(* Schneider Machine Expert - Basic project TMA0070_BOTTOM CASE SCREWING, file version 2.8.0.0 *)
(* ProjectInformations: Name=New project *)

HARDWARE
  Cpu 0: TM221CE16T
  EthernetConfiguration: NetworkName=M221, IpAllocationMode=FixedAddress, IpAddress=192.168.0.150, SubnetMask=255.255.255.0
  SerialLineConfiguration: Baud=Baud19200, Parity=ParityEven, DataBits=DataBits8, StopBits=StopBits1, PhysicalMedium=PhysicalMediumRs485, TransmissionMode=TransmissionModeModbusRtu, SlaveId=1, Addressing=SlaveAddressing
  MastTask: UsePeriodScanMode=false, PeriodScan=100
  FastTask: Period=255
  CpuBehavior: StartingMode=StartAsPreviousState, AutoSaveRamOnEeprom=true, WatchdogPeriod=250

SYMBOLS  (address, symbol, comment, settings)
  %M20      IB_ESTOP
  %M21      IB_CYL  "TURUNSTART"
  %M23      IB_TIMER
  %M27      VALID_BARCODE
  %M28      INVALID_BARCODE
  %M29      IB_TRIGGER_KEYENCE
  %M32      MACHINE_RUNNING
  %M33      ERROR_BARCODE
  %M34      SAFETY_TRIGGER
  %M35      TURUNDONE_SENSOR_TURUN
  %M80      PASS
  %TM0        [Preset=2, Base=OneSecond]
  %TM1        [Preset=2, Base=OneSecond]
  %I0.0     ESTOP
  %I0.1     START_PB
  %I0.2     RESET_PB
  %I0.3     CURTAIN  "CURTAIN SENSOR"
  %I0.4     C_NEWTON  "CHECK OUTX LOAD CELL"
  %I0.5     TIMER  "TIMER DONE"
  %I0.6     RS_CYL_UP
  %I0.7     RS_CYL_DOWN
  %Q0.0     CYL_PRESS
  %Q0.1     START_TIIMER
  %Q0.2     TRIGGER_KEYENCE
  %Q0.3     RED_LIGHT
  %Q0.4     YELLOW_LIGHT_
  %Q0.5     GREEN_LIGHT
  %IW0.0      [Type=Type_0_10V, Scope=Scope_Normal, Minimum=0, Maximum=1000]

POU SEQUENCE
  (* SectionNumber=1 *)

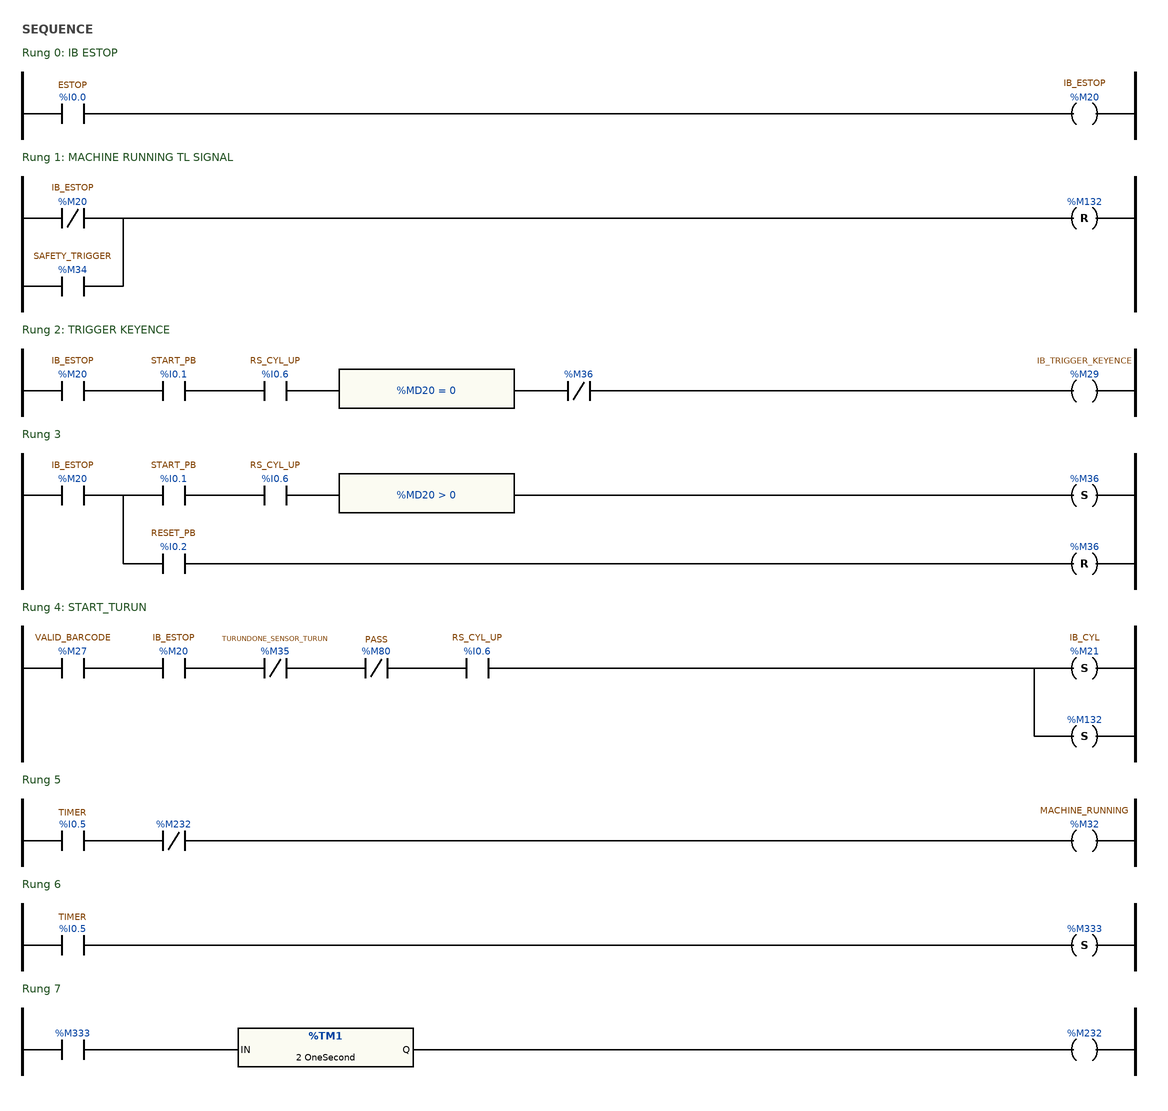

// Rung 0: IB ESTOP
  LD %I0.0                (* ESTOP *)
  ST %M20                 (* IB_ESTOP *)
  // as ST:
  //   IB_ESTOP := ESTOP;

// Rung 1: MACHINE RUNNING TL SIGNAL
  LDN %M20                (* IB_ESTOP *)
  OR %M34                 (* SAFETY_TRIGGER *)
  R %M132
  // as ST:
  //   IF NOT IB_ESTOP OR SAFETY_TRIGGER THEN %M132 := FALSE; END_IF;

// Rung 2: TRIGGER KEYENCE
  LD %M20                 (* IB_ESTOP *)
  AND %I0.1               (* START_PB *)
  AND %I0.6               (* RS_CYL_UP *)
  AND [ %MD20 = 0 ]
  ANDN %M36
  ST %M29                 (* IB_TRIGGER_KEYENCE *)
  // as ST:
  //   IB_TRIGGER_KEYENCE := IB_ESTOP AND START_PB AND RS_CYL_UP AND %MD20 = 0 AND NOT %M36;

// Rung 3
  LD %M20                 (* IB_ESTOP *)
  MPS
  AND %I0.1               (* START_PB *)
  AND %I0.6               (* RS_CYL_UP *)
  AND [ %MD20 > 0 ]
  S %M36
  MPP
  AND %I0.2               (* RESET_PB *)
  R %M36
  // as ST:
  //   IF IB_ESTOP AND START_PB AND RS_CYL_UP AND %MD20 > 0 THEN %M36 := TRUE; END_IF;
  //   IF IB_ESTOP AND RESET_PB THEN %M36 := FALSE; END_IF;

// Rung 4: START_TURUN
  LD %M27                 (* VALID_BARCODE *)
  AND %M20                (* IB_ESTOP *)
  ANDN %M35               (* TURUNDONE_SENSOR_TURUN *)
  ANDN %M80               (* PASS *)
  AND %I0.6               (* RS_CYL_UP *)
  S %M21                  (* IB_CYL *)
  S %M132
  // as ST:
  //   IF VALID_BARCODE AND IB_ESTOP AND NOT TURUNDONE_SENSOR_TURUN AND NOT PASS AND RS_CYL_UP THEN IB_CYL := TRUE; END_IF;
  //   IF VALID_BARCODE AND IB_ESTOP AND NOT TURUNDONE_SENSOR_TURUN AND NOT PASS AND RS_CYL_UP THEN %M132 := TRUE; END_IF;

// Rung 5
  LD %I0.5                (* TIMER *)
  ANDN %M232
  ST %M32                 (* MACHINE_RUNNING *)
  // as ST:
  //   MACHINE_RUNNING := TIMER AND NOT %M232;

// Rung 6
  LD %I0.5                (* TIMER *)
  S %M333
  // as ST:
  //   IF TIMER THEN %M333 := TRUE; END_IF;

// Rung 7
  BLK %TM1
  LD %M333
  IN
  OUT_BLK
  LD Q
  ST %M232
  END_BLK
  // as ST:
  //   %TM1(IN := %M333);
  //   %M232 := %TM1.Q;

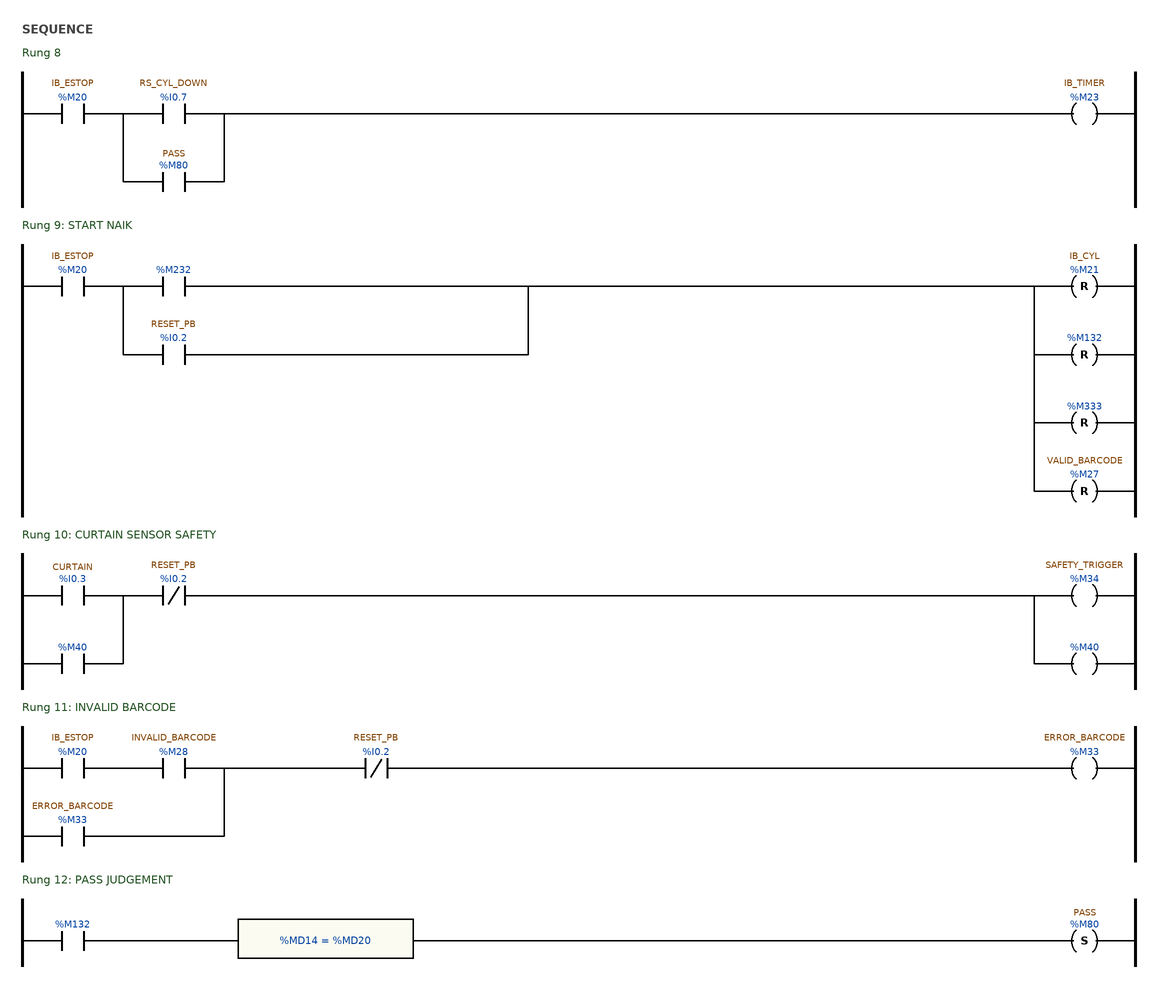

// Rung 8
  LD %M20                 (* IB_ESTOP *)
  AND( %I0.7              (* RS_CYL_DOWN *)
  OR %M80                 (* PASS *)
  )
  ST %M23                 (* IB_TIMER *)
  // as ST:
  //   IB_TIMER := IB_ESTOP AND (RS_CYL_DOWN OR PASS);

// Rung 9: START NAIK
  LD %M20                 (* IB_ESTOP *)
  AND( %M232
  OR %I0.2                (* RESET_PB *)
  )
  R %M21                  (* IB_CYL *)
  R %M132
  R %M333
  R %M27                  (* VALID_BARCODE *)
  // as ST:
  //   IF IB_ESTOP AND (%M232 OR RESET_PB) THEN IB_CYL := FALSE; END_IF;
  //   IF IB_ESTOP AND (%M232 OR RESET_PB) THEN %M132 := FALSE; END_IF;
  //   IF IB_ESTOP AND (%M232 OR RESET_PB) THEN %M333 := FALSE; END_IF;
  //   IF IB_ESTOP AND (%M232 OR RESET_PB) THEN VALID_BARCODE := FALSE; END_IF;

// Rung 10: CURTAIN SENSOR SAFETY
  LD %I0.3                (* CURTAIN *)
  OR %M40
  ANDN %I0.2              (* RESET_PB *)
  ST %M34                 (* SAFETY_TRIGGER *)
  ST %M40
  // as ST:
  //   SAFETY_TRIGGER := (CURTAIN OR %M40) AND NOT RESET_PB;
  //   %M40 := (CURTAIN OR %M40) AND NOT RESET_PB;

// Rung 11: INVALID BARCODE
  LD %M20                 (* IB_ESTOP *)
  AND %M28                (* INVALID_BARCODE *)
  OR %M33                 (* ERROR_BARCODE *)
  ANDN %I0.2              (* RESET_PB *)
  ST %M33                 (* ERROR_BARCODE *)
  // as ST:
  //   ERROR_BARCODE := (IB_ESTOP AND INVALID_BARCODE OR ERROR_BARCODE) AND NOT RESET_PB;

// Rung 12: PASS JUDGEMENT
  LD %M132
  AND [ %MD14 = %MD20 ]
  S %M80                  (* PASS *)
  // as ST:
  //   IF %M132 AND %MD14 = %MD20 THEN PASS := TRUE; END_IF;

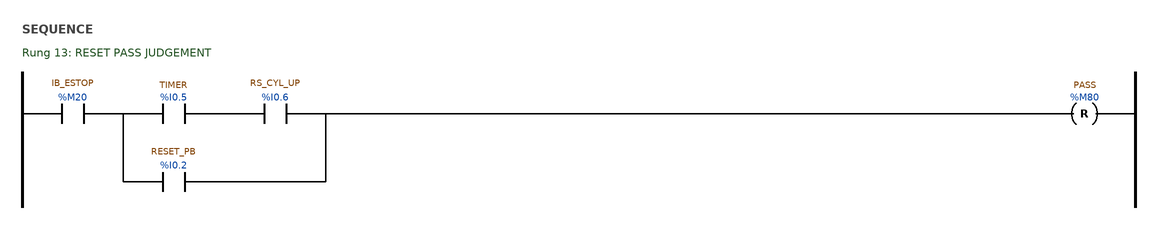

// Rung 13: RESET PASS JUDGEMENT
  LD %M20                 (* IB_ESTOP *)
  AND( %I0.5              (* TIMER *)
  AND %I0.6               (* RS_CYL_UP *)
  OR %I0.2                (* RESET_PB *)
  )
  R %M80                  (* PASS *)
  // as ST:
  //   IF IB_ESTOP AND (TIMER AND RS_CYL_UP OR RESET_PB) THEN PASS := FALSE; END_IF;

POU I/0
  (* SectionNumber=2 *)

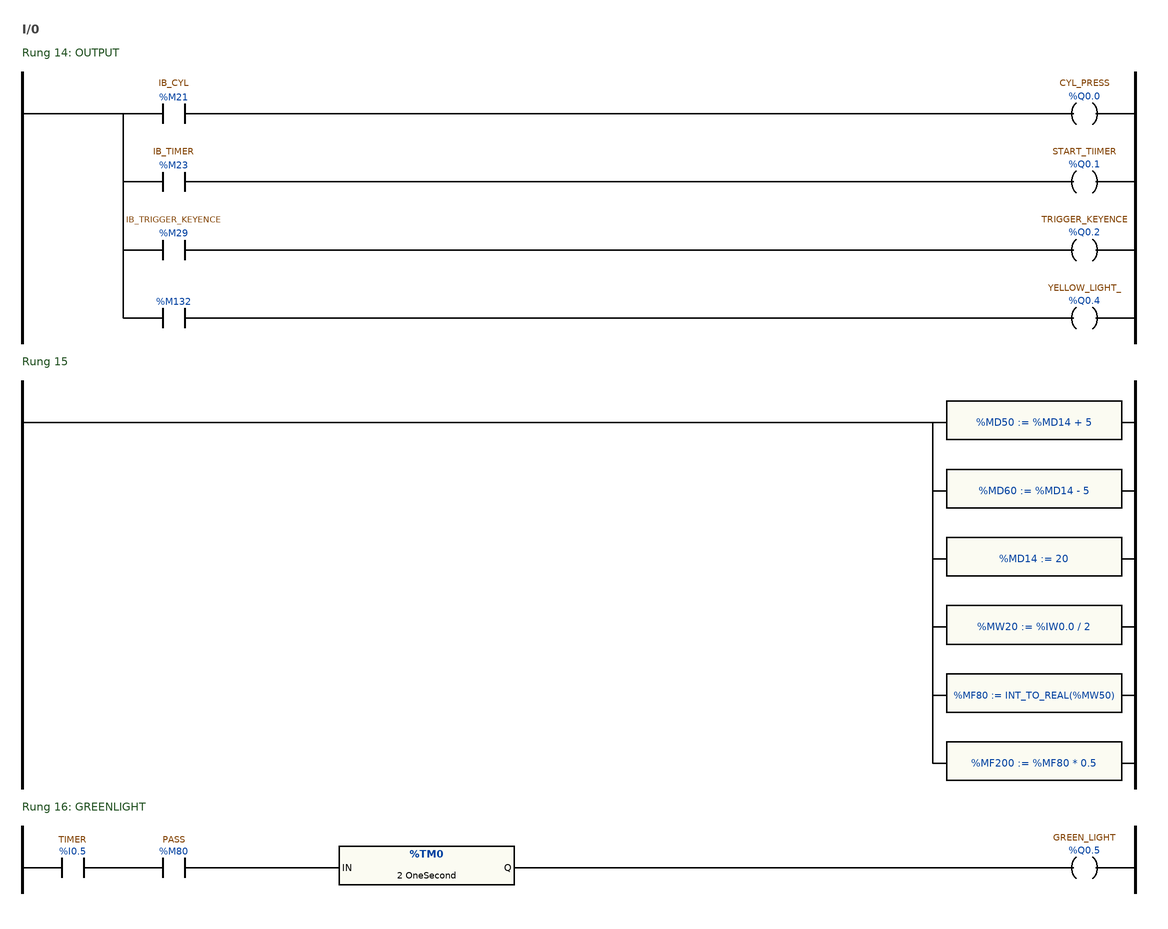

// Rung 14: OUTPUT
  LD 1
  MPS
  AND %M21                (* IB_CYL *)
  ST %Q0.0                (* CYL_PRESS *)
  MRD
  AND %M23                (* IB_TIMER *)
  ST %Q0.1                (* START_TIIMER *)
  MRD
  AND %M29                (* IB_TRIGGER_KEYENCE *)
  ST %Q0.2                (* TRIGGER_KEYENCE *)
  MPP
  AND %M132
  ST %Q0.4                (* YELLOW_LIGHT_ *)
  // as ST:
  //   CYL_PRESS := IB_CYL;
  //   START_TIIMER := IB_TIMER;
  //   TRIGGER_KEYENCE := IB_TRIGGER_KEYENCE;
  //   YELLOW_LIGHT_ := %M132;

// Rung 15
  LD 1
  [ %MD50 := %MD14 + 5 ]
  [ %MD60 := %MD14 - 5 ]
  [ %MD14 := 20 ]
  [ %MW20 := %IW0.0 / 2 ]
  [ %MF80 := INT_TO_REAL ( %MW50 ) ]
  [ %MF200 := %MF80 * 0.5 ]
  // as ST:
  //   %MD50 := %MD14 + 5;
  //   %MD60 := %MD14 - 5;
  //   %MD14 := 20;
  //   %MW20 := %IW0.0 / 2;
  //   %MF80 := INT_TO_REAL ( %MW50 );
  //   %MF200 := %MF80 * 0.5;

// Rung 16: GREENLIGHT
  BLK %TM0
  LD %I0.5                (* TIMER *)
  AND %M80                (* PASS *)
  IN
  OUT_BLK
  LD Q
  ST %Q0.5                (* GREEN_LIGHT *)
  END_BLK
  // as ST:
  //   %TM0(IN := TIMER AND PASS);
  //   GREEN_LIGHT := %TM0.Q;
